FUNCTION_BLOCK FB_CycleInit
VAR_INPUT
	xStart : BOOL;
	xStop : BOOL;
	xReset:BOOL;
END_VAR
VAR_OUTPUT
	fbRtrigStart:R_trig;
	xBusy:BOOL;
	iEtape:INT;
END_VAR
VAR
	fbEtape:FB_Etape;
END_VAR

fbEtape.mActualisation(stParam.stStatus.xModePasAPas,fbBtn.xNextPas);

fbRtrigStart(clk:=fbBtn.xStart);

IF xReset THEN
	fbEtape.piVal:=0;
	xBusy:=FALSE;
END_IF

CASE fbEtape.iNo OF
	0:fbEtape.psMess:='Init | Wait';
		IF xStart THEN
			fbEtape.piVal:=99;
		END_IF
	
	
	99: fbEtape.psMess:='Init | Reset on Actuators and Motor';
		IF  stParam.stStatus.xHomingDone=TRUE THEN
			fbEtape.piSVal:=400;
		ELSE
			fbEtape.piSVal:=100;
		END_IF
	100: fbEtape.psMess:='Start Homing X';
			fbEtape.tTimeQ:=T#100MS;
			fbEtape.piSVal:=101;
	101:fbEtape.psMess:='Init | Wait 100MS';
		IF fbEtape.xTimeQ THEN
			fbEtape.piSVal:=102;
		END_IF
	102: fbEtape.psMess:='Init | Waiting for Homing Axis X';
		IF NOT fbMotorX.mcHome.Active AND NOT fbBtn.xHomingPosReached THEN
			fbEtape.piVal:=200;
		END_IF
		
	200:fbEtape.psMess:='Init | Start Homing Axis Y';
		fbEtape.piVal:=201;
		fbEtape.tTimeQ:=T#100MS;
	201:fbEtape.psMess:='Init | Wait 100MS';
		IF fbEtape.xTimeQ THEN
			fbEtape.piSVal:=202;
		END_IF
	202: fbEtape.psMess:='Init | Waiting for Homing Axis Y';
		IF NOT fbMotorY.mcHome.Active AND NOT fbBtn.xHomingPosReached THEN
			fbEtape.piVal:=300;
		END_IF
		
	300:fbEtape.psMess:='Init | Start Homing Axis Z';
		fbEtape.piVal:=301;
		fbEtape.tTimeQ:=T#100MS;
	301:fbEtape.psMess:='Init | Wait 100MS';
		IF fbEtape.xTimeQ THEN
			fbEtape.piSVal:=302;
		END_IF
	302: fbEtape.psMess:='Init | Waiting for Homing Axis Z';
		IF NOT fbMotorZ.mcHome.Active AND NOT fbBtn.xHomingPosReached THEN
			fbEtape.piVal:=400;
			stParam.stStatus.xHomingDone:=TRUE;
		END_IF
		
		
	400:fbEtape.psMess:='Init | Init Actor1';
		IF  fbAct1.xInInPos AND stParam.stMachine.stPosition0.Initialized=FALSE THEN
			fbEtape.piSVal:=500;
		ELSIF  fbAct1.xInInPos AND stParam.stMachine.stPosition0.Initialized=TRUE THEN
			fbEtape.piSVal:=999;
		END_IF
		
	500:fbEtape.psMess:='Init | Init Home Position';
		IF  fbBtn.xSetHomePos THEN
			stParam.stMachine.stPosition0.Initialized:=TRUE;
			stParam.stMachine.stPosition0.PosX:=fbMotorX.fbAxisRef.NcToPlc.ActPos;
			stParam.stMachine.stPosition0.PosY:=fbMotorY.fbAxisRef.NcToPlc.ActPos;
			fbEtape.piSVal:=999;
		END_IF
		
		
	
	999:fbEtape.psMess:='Init | Finished';
		IF (xStop) THEN
		fbEtape.piSVal:=0;
	END_IF
END_CASE

xBusy:=fbEtape.iNo<>0;
iEtape:=fbEtape.iNo;

END_FUNCTION_BLOCK

(* stored: Version 1.1.0.1, ProductVersion 3.1.4020.12
   POU FB_CycleInit: Id {78f8b3c7-c7ef-4e76-a081-037ca3472bc0}, SpecialFunc None *)
